// TIA Portal V18 export
// export: Created 2026-03-12T16:04:36.0951066Z, ExportSetting WithDefaults, DisplayName Totally Integrated Automation Portal, DisplayVersion V18 Update 5, DisplayName TIA Portal Openness, DisplayVersion V18 Update 5, DisplayName TIA Portal Version Control Interface, DisplayVersion V18, DisplayName SINAMICS Startdrive Advanced, DisplayVersion V18, DisplayName SINAMICS Startdrive G130, G150, S120, S150, SINAMICS MV, S210, DisplayVersion V18, DisplayName SINAMICS Startdrive G110M, G120, G120C, G120D, G120P, G115D, DisplayVersion V18, DisplayName STEP 7 Professional, DisplayVersion V18 Update 5, DisplayName STEP 7 Safety, DisplayVersion V18, DisplayName WinCC Professional, DisplayVersion V18 Update 5
FUNCTION_BLOCK "FB PROCESSO_AUTO_ELEVATORIA"   // FB38, LAD
{ S7_Optimized_Access := 'TRUE' }
VERSION : 0.1
// stored: AutoNumber true, IsIECCheckEnabled false, IsRetainMemResEnabled false, MemoryReserve 100, SetENOAutomatically false, UDAEnableTagReadback false
   VAR_INPUT
      INPUT_HABILITA_PAR : Bool;
      INPUT_REMOTO_AUTO_A : Bool;
      INPUT_REMOTO_AUTO_B : Bool;
      INPUT_COMANDO_ALTERNANCIA_ATIVO : Bool;
      INPUT_FALHA_BOMBA_A : Bool;
      INPUT_FALHA_BOMBA_B : Bool;
      INPUT_CADASTRO_TEMPO_LIGADO_A : Real;
      INPUT_CADASTRO_TEMPO_LIGADO_B : Real;
      INPUT_STATUS_SENSOR : Real;
      INPUT_CADASTRO_LIGA_A : Real;
      INPUT_CADASTRO_DESLIGA_A : Real;
      INPUT_CADASTRO_LIGA_B : Real;
      INPUT_CADASTRO_DESLIGA_B : Real;
   END_VAR
   VAR_OUTPUT
      HORA_ALTERNANCIA_A : Real;
      HORA_ALTERNANCIA_B : Real;
      HABILITA_LIGA_BOMBA_A : Bool;
      HABILITA_LIGA_BOMBA_B : Bool;
   END_VAR
   VAR
      "FB CONTADOR_A" { S7_SetPoint := 'True'} : "FB CONTADOR";
      "FB CONTADOR_B" { S7_SetPoint := 'True'} : "FB CONTADOR";
   END_VAR
   VAR_TEMP
      "ALTERNANCIA_ATIVA_A_&_B" : Bool;
      LIGA_ALTERNANCIA_A : Bool;
      LIGA_ALTERNANCIA_B : Bool;
      HABILITA_LIGA_COMPARATIVO_A : Bool;
      HABILITA_LIGA_COMPARATIVO_B : Bool;
   END_VAR
   VAR_TEMP   // added for the SCL form of the ladder/FBD networks
      _w1 : Bool;
   END_VAR
BEGIN

REGION Network 1: Alternância/Rotatividade de bomba Principal
   // Conforme alternância habilitada, a bomba principal e reserva trabalharão intercaladas baseando-se no tempos cadastrados pela operação.
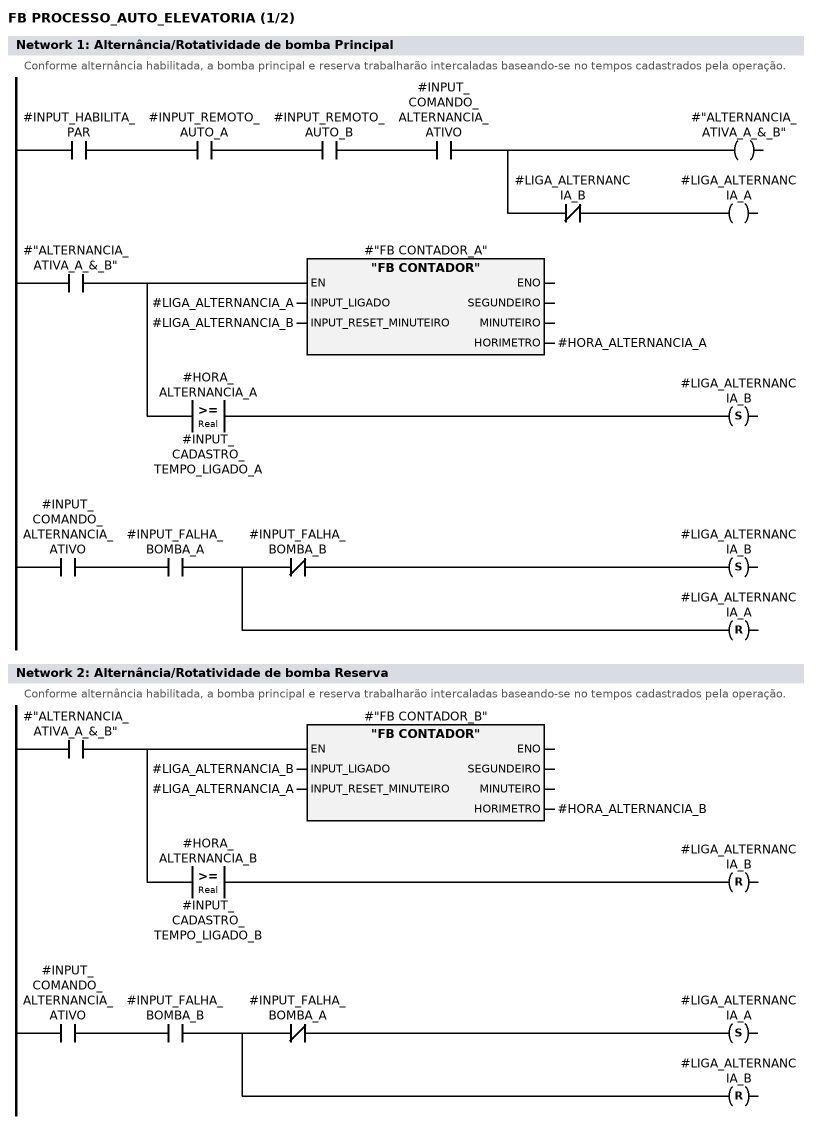
   RUNG wire#powerrail
      Contact( #INPUT_HABILITA_PAR )
      Contact( #INPUT_REMOTO_AUTO_A )
      Contact( #INPUT_REMOTO_AUTO_B )
      Contact( #INPUT_COMANDO_ALTERNANCIA_ATIVO )
      wire#w1
      Coil( #"ALTERNANCIA_ATIVA_A_&_B" )
   END_RUNG
   RUNG wire#w1
      I_Contact( #LIGA_ALTERNANCIA_B )
      Coil( #LIGA_ALTERNANCIA_A )
   END_RUNG
   RUNG wire#powerrail
      Contact( #"ALTERNANCIA_ATIVA_A_&_B" )
      wire#w2
      #"FB CONTADOR_A"(INPUT_LIGADO := #LIGA_ALTERNANCIA_A, INPUT_RESET_MINUTEIRO := #LIGA_ALTERNANCIA_B, SEGUNDEIRO =>, MINUTEIRO =>, HORIMETRO => #HORA_ALTERNANCIA_A)
   END_RUNG
   RUNG wire#w2
      { S7_Templates := "SrcType := Real" } GE_Contact(in1 := #HORA_ALTERNANCIA_A, in2 := #INPUT_CADASTRO_TEMPO_LIGADO_A)
      S_Coil( #LIGA_ALTERNANCIA_B )
   END_RUNG
   RUNG wire#powerrail
      Contact( #INPUT_COMANDO_ALTERNANCIA_ATIVO )
      Contact( #INPUT_FALHA_BOMBA_A )
      wire#w3
      I_Contact( #INPUT_FALHA_BOMBA_B )
      S_Coil( #LIGA_ALTERNANCIA_B )
   END_RUNG
   RUNG wire#w3
      R_Coil( #LIGA_ALTERNANCIA_A )
   END_RUNG
   // the same network as SCL:
   #"ALTERNANCIA_ATIVA_A_&_B" := #INPUT_HABILITA_PAR AND #INPUT_REMOTO_AUTO_A AND #INPUT_REMOTO_AUTO_B AND #INPUT_COMANDO_ALTERNANCIA_ATIVO;
   #LIGA_ALTERNANCIA_A := #"ALTERNANCIA_ATIVA_A_&_B" AND NOT #LIGA_ALTERNANCIA_B;
   IF #"ALTERNANCIA_ATIVA_A_&_B" THEN
       #"FB CONTADOR_A"(INPUT_LIGADO := #LIGA_ALTERNANCIA_A,   // "FB CONTADOR"
                        INPUT_RESET_MINUTEIRO := #LIGA_ALTERNANCIA_B,
                        HORIMETRO => #HORA_ALTERNANCIA_A);
   END_IF;
   IF #"ALTERNANCIA_ATIVA_A_&_B" AND (#HORA_ALTERNANCIA_A >= #INPUT_CADASTRO_TEMPO_LIGADO_A) THEN
       #LIGA_ALTERNANCIA_B := TRUE;
   END_IF;
   #_w1 := #INPUT_COMANDO_ALTERNANCIA_ATIVO AND #INPUT_FALHA_BOMBA_A;
   IF #_w1 AND NOT #INPUT_FALHA_BOMBA_B THEN #LIGA_ALTERNANCIA_B := TRUE; END_IF;
   IF #_w1 THEN #LIGA_ALTERNANCIA_A := FALSE; END_IF;
END_REGION

REGION Network 2: Alternância/Rotatividade de bomba Reserva
   // Conforme alternância habilitada, a bomba principal e reserva trabalharão intercaladas baseando-se no tempos cadastrados pela operação.
   RUNG wire#powerrail
      Contact( #"ALTERNANCIA_ATIVA_A_&_B" )
      wire#w1
      #"FB CONTADOR_B"(INPUT_LIGADO := #LIGA_ALTERNANCIA_B, INPUT_RESET_MINUTEIRO := #LIGA_ALTERNANCIA_A, SEGUNDEIRO =>, MINUTEIRO =>, HORIMETRO => #HORA_ALTERNANCIA_B)
   END_RUNG
   RUNG wire#w1
      { S7_Templates := "SrcType := Real" } GE_Contact(in1 := #HORA_ALTERNANCIA_B, in2 := #INPUT_CADASTRO_TEMPO_LIGADO_B)
      R_Coil( #LIGA_ALTERNANCIA_B )
   END_RUNG
   RUNG wire#powerrail
      Contact( #INPUT_COMANDO_ALTERNANCIA_ATIVO )
      Contact( #INPUT_FALHA_BOMBA_B )
      wire#w2
      I_Contact( #INPUT_FALHA_BOMBA_A )
      S_Coil( #LIGA_ALTERNANCIA_A )
   END_RUNG
   RUNG wire#w2
      R_Coil( #LIGA_ALTERNANCIA_B )
   END_RUNG
   // the same network as SCL:
   IF #"ALTERNANCIA_ATIVA_A_&_B" THEN
       #"FB CONTADOR_B"(INPUT_LIGADO := #LIGA_ALTERNANCIA_B,   // "FB CONTADOR"
                        INPUT_RESET_MINUTEIRO := #LIGA_ALTERNANCIA_A,
                        HORIMETRO => #HORA_ALTERNANCIA_B);
   END_IF;
   IF #"ALTERNANCIA_ATIVA_A_&_B" AND (#HORA_ALTERNANCIA_B >= #INPUT_CADASTRO_TEMPO_LIGADO_B) THEN
       #LIGA_ALTERNANCIA_B := FALSE;
   END_IF;
   #_w1 := #INPUT_COMANDO_ALTERNANCIA_ATIVO AND #INPUT_FALHA_BOMBA_B;
   IF #_w1 AND NOT #INPUT_FALHA_BOMBA_A THEN #LIGA_ALTERNANCIA_A := TRUE; END_IF;
   IF #_w1 THEN #LIGA_ALTERNANCIA_B := FALSE; END_IF;
END_REGION

REGION Network 3: Condições para Modo Automático Bomba A
   // - Caso o nível da elevatória seja inferior ao setpoint cadastrado para desligar a bomba, esta desligará. 
   // - Caso o nível da elevatória seja superior ao setpoint cadastrado para ligar, esta irá ligar.
   // - Se HABILITA_LIGA_COMPARATIVO for 1 então nível habilita liga, e Intertravamento "1" então Rotatividade Habilitada, a bomba só ira ligar com a condição de alternancia "1".
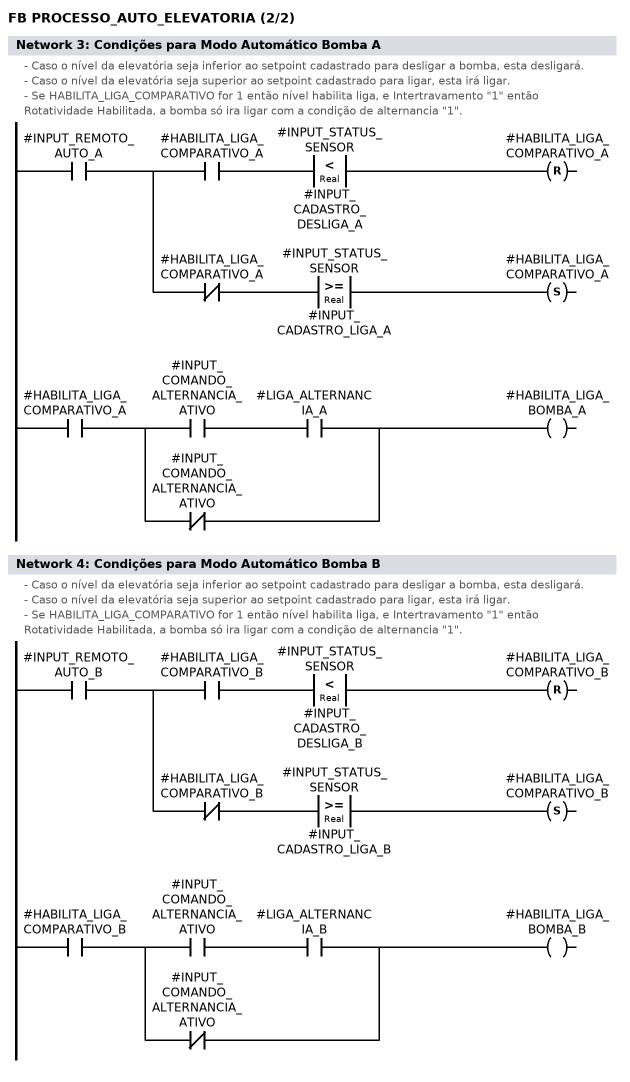
   RUNG wire#powerrail
      Contact( #INPUT_REMOTO_AUTO_A )
      wire#w1
      Contact( #HABILITA_LIGA_COMPARATIVO_A )
      { S7_Templates := "SrcType := Real" } LT_Contact(in1 := #INPUT_STATUS_SENSOR, in2 := #INPUT_CADASTRO_DESLIGA_A)
      R_Coil( #HABILITA_LIGA_COMPARATIVO_A )
   END_RUNG
   RUNG wire#w1
      I_Contact( #HABILITA_LIGA_COMPARATIVO_A )
      { S7_Templates := "SrcType := Real" } GE_Contact(in1 := #INPUT_STATUS_SENSOR, in2 := #INPUT_CADASTRO_LIGA_A)
      S_Coil( #HABILITA_LIGA_COMPARATIVO_A )
   END_RUNG
   RUNG wire#powerrail
      Contact( #HABILITA_LIGA_COMPARATIVO_A )
      wire#w2
      Contact( #INPUT_COMANDO_ALTERNANCIA_ATIVO )
      Contact( #LIGA_ALTERNANCIA_A )
      wire#w3
      Coil( #HABILITA_LIGA_BOMBA_A )
   END_RUNG
   RUNG wire#w2
      I_Contact( #INPUT_COMANDO_ALTERNANCIA_ATIVO )
   END_RUNG wire#w3
   // the same network as SCL:
   IF #INPUT_REMOTO_AUTO_A AND #HABILITA_LIGA_COMPARATIVO_A AND (#INPUT_STATUS_SENSOR < #INPUT_CADASTRO_DESLIGA_A) THEN
       #HABILITA_LIGA_COMPARATIVO_A := FALSE;
   END_IF;
   IF #INPUT_REMOTO_AUTO_A AND NOT #HABILITA_LIGA_COMPARATIVO_A AND (#INPUT_STATUS_SENSOR >= #INPUT_CADASTRO_LIGA_A) THEN
       #HABILITA_LIGA_COMPARATIVO_A := TRUE;
   END_IF;
   #HABILITA_LIGA_BOMBA_A := #HABILITA_LIGA_COMPARATIVO_A AND ((#INPUT_COMANDO_ALTERNANCIA_ATIVO AND #LIGA_ALTERNANCIA_A) OR NOT #INPUT_COMANDO_ALTERNANCIA_ATIVO);
END_REGION

REGION Network 4: Condições para Modo Automático Bomba B
   // - Caso o nível da elevatória seja inferior ao setpoint cadastrado para desligar a bomba, esta desligará. 
   // - Caso o nível da elevatória seja superior ao setpoint cadastrado para ligar, esta irá ligar.
   // - Se HABILITA_LIGA_COMPARATIVO for 1 então nível habilita liga, e Intertravamento "1" então Rotatividade Habilitada, a bomba só ira ligar com a condição de alternancia "1".
   RUNG wire#powerrail
      Contact( #INPUT_REMOTO_AUTO_B )
      wire#w1
      Contact( #HABILITA_LIGA_COMPARATIVO_B )
      { S7_Templates := "SrcType := Real" } LT_Contact(in1 := #INPUT_STATUS_SENSOR, in2 := #INPUT_CADASTRO_DESLIGA_B)
      R_Coil( #HABILITA_LIGA_COMPARATIVO_B )
   END_RUNG
   RUNG wire#w1
      I_Contact( #HABILITA_LIGA_COMPARATIVO_B )
      { S7_Templates := "SrcType := Real" } GE_Contact(in1 := #INPUT_STATUS_SENSOR, in2 := #INPUT_CADASTRO_LIGA_B)
      S_Coil( #HABILITA_LIGA_COMPARATIVO_B )
   END_RUNG
   RUNG wire#powerrail
      Contact( #HABILITA_LIGA_COMPARATIVO_B )
      wire#w2
      Contact( #INPUT_COMANDO_ALTERNANCIA_ATIVO )
      Contact( #LIGA_ALTERNANCIA_B )
      wire#w3
      Coil( #HABILITA_LIGA_BOMBA_B )
   END_RUNG
   RUNG wire#w2
      I_Contact( #INPUT_COMANDO_ALTERNANCIA_ATIVO )
   END_RUNG wire#w3
   // the same network as SCL:
   IF #INPUT_REMOTO_AUTO_B AND #HABILITA_LIGA_COMPARATIVO_B AND (#INPUT_STATUS_SENSOR < #INPUT_CADASTRO_DESLIGA_B) THEN
       #HABILITA_LIGA_COMPARATIVO_B := FALSE;
   END_IF;
   IF #INPUT_REMOTO_AUTO_B AND NOT #HABILITA_LIGA_COMPARATIVO_B AND (#INPUT_STATUS_SENSOR >= #INPUT_CADASTRO_LIGA_B) THEN
       #HABILITA_LIGA_COMPARATIVO_B := TRUE;
   END_IF;
   #HABILITA_LIGA_BOMBA_B := #HABILITA_LIGA_COMPARATIVO_B AND ((#INPUT_COMANDO_ALTERNANCIA_ATIVO AND #LIGA_ALTERNANCIA_B) OR NOT #INPUT_COMANDO_ALTERNANCIA_ATIVO);
END_REGION
END_FUNCTION_BLOCK
